// Block: A0302_OB30_Status

DATA_BLOCK A0302_OB30_Status
VERSION : 0.1
   NON_RETAIN
   VAR
      RETVAL_SET_CINT_Low : Int;
      RETVAL_SET_CINT_High : Int;
      RETVAL_QRY_CINT_Low : Int;
      RETVAL_QRY_CINT_High : Int;
      QRT_OB30_Low_CYCLE : UDInt;
      QRT_OB30_Low_PHASE : UDInt;
      QRT_OB30_Low_STATUS : Word;
      QRT_OB30_High_CYCLE : UDInt;
      QRT_OB30_High_PHASE : UDInt;
      QRT_OB30_High_STATUS : Word;
      OB30_Low : Bool;
      OB30_High : Bool;
   END_VAR

BEGIN
   // No initialization required
END_DATA_BLOCK
